FUNCTION Convert_UDINT_TO_REAL : Hresult
VAR_INPUT
	in : UDINT;
	out : REFERENCE TO REAL;
END_VAR
VAR
	converted : REAL;
END_VAR

converted := UDINT_TO_REAL(in);

IF (REAL_TO_UDINT(converted) <> in) THEN
	Convert_UDINT_TO_REAL := INCOMPATIBLE;
	RETURN;
END_IF

out := converted;

END_FUNCTION

(* stored: Version 1.1.0.1, ProductVersion 3.1.4024.12
   POU Convert_UDINT_TO_REAL: Id {c587dd12-d0d5-437e-ae22-f89fa7db6af4}, SpecialFunc None *)
